FUNCTION_BLOCK Sensor_NOpen IMPLEMENTS I_Sensor
VAR
	bInput AT %I* : BOOL;
END_VAR

PROPERTY isActive : BOOL
GET
isActive:=bInput;
END_GET
END_PROPERTY

PROPERTY notActive : BOOL
GET
notActive:= NOT bInput;
END_GET
END_PROPERTY

END_FUNCTION_BLOCK

(* stored: Version 1.1.0.1, ProductVersion 3.1.4024.12
   POU Sensor_NOpen: Id {8107bbcb-a92a-48f3-add1-ef65f3e406fd}, SpecialFunc None
   Property isActive: Id {5c5bc8ee-b49a-4fab-818d-30d504b6f969}
   Get Get: Id {f4df5b59-7268-4521-8f4b-0a81849c27ce}
   Property notActive: Id {894eb1bd-ffb9-4748-b909-0d921fdeea90}
   Get Get: Id {24918f9a-9eb3-472a-8f2a-8126c542b497} *)
